METHOD PUBLIC TestTryGetKeyUint
VAR
    jsonDeserializer : JsonDeserializer;
    json : STRING := '{"data":12345}';
    out : UINT;
	feedback : DeserializerFeedback;
    expected : UINT := 12345;
END_VAR
TEST('TestTryGetKeyUint');

jsonDeserializer.TryLoad(json);
jsonDeserializer.TryGetKeyUint('data', out, feedback);

AssertEquals(
    Expected := expected,
    Actual := out,
    Message := 'Did not produce the expected UINT value from JSON'
);

TEST_FINISHED();
END_METHOD

METHOD PUBLIC TestTryGetKeyUlint
VAR
    jsonDeserializer : JsonDeserializer;
    json : STRING := '{"data":9223372036854775807}';
    out : ULINT;
	feedback : DeserializerFeedback;
    expected : ULINT := 9223372036854775807;
END_VAR
TEST('TestTryGetKeyUlint');

jsonDeserializer.TryLoad(json);
jsonDeserializer.TryGetKeyUlint('data', out, feedback);

AssertEquals(
    Expected := expected,
    Actual := out,
    Message := 'Did not produce the expected ULINT value from JSON'
);

TEST_FINISHED();
END_METHOD

METHOD PUBLIC TestTryGetKeyUsint
VAR
    jsonDeserializer : JsonDeserializer;
    json : STRING := '{"data":123}';
    out : USINT;
	feedback : DeserializerFeedback;
    expected : USINT := 123;
END_VAR
TEST('TestTryGetKeyUsint');

jsonDeserializer.TryLoad(json);
jsonDeserializer.TryGetKeyUsint('data', out, feedback);

AssertEquals(
    Expected := expected,
    Actual := out,
    Message := 'Did not produce the expected USINT value from JSON'
);

TEST_FINISHED();
END_METHOD

METHOD PUBLIC TestTryGetKeyWord
VAR
    jsonDeserializer : JsonDeserializer;
    json : STRING := '{"data":12345}';
    out : WORD;
	feedback : DeserializerFeedback;
    expected : WORD := 12345;
END_VAR
TEST('TestTryGetKeyWord');

jsonDeserializer.TryLoad(json);
jsonDeserializer.TryGetKeyWord('data', out, feedback);

AssertEquals(
    Expected := expected,
    Actual := out,
    Message := 'Did not produce the expected WORD value from JSON'
);

TEST_FINISHED();
END_METHOD

METHOD PUBLIC TestTryGetLint
VAR
    jsonDeserializer : JsonDeserializer;
    json : STRING := '9223372036854775807';
    out : LINT;
	feedback : DeserializerFeedback;
    expected : LINT := 9223372036854775807;
END_VAR
TEST('TestTryGetLint');

jsonDeserializer.TryLoad(json);
jsonDeserializer.TryGetLint(out, feedback);

AssertEquals(
    Expected := expected,
    Actual := out,
    Message := 'Did not produce the expected LINT value from JSON'
);

TEST_FINISHED();
END_METHOD

METHOD PUBLIC TestTryGetLreal
VAR
    jsonDeserializer : JsonDeserializer;
    json : STRING := '123456.789';
    out : LREAL;
	feedback : DeserializerFeedback;
    expected : LREAL := 123456.789;
END_VAR
TEST('TestTryGetLreal');

jsonDeserializer.TryLoad(json);
jsonDeserializer.TryGetLreal(out, feedback);

AssertEquals(
    Expected := expected,
    Actual := out,
    Message := 'Did not produce the expected LREAL value from JSON'
);

TEST_FINISHED();
END_METHOD

METHOD PUBLIC TestTryGetLtime
VAR
    jsonDeserializer : JsonDeserializer;
    json : STRING := '"LTIME#100d2h30m40s500ms600us700ns"';
    out : LTIME;
	feedback : DeserializerFeedback;
    expected : LTIME := LTIME#100D2H30M40S500MS600US700NS;
END_VAR
TEST('TestTryGetLtime');

jsonDeserializer.TryLoad(json);
jsonDeserializer.TryGetLtime(out, feedback);

AssertEquals(
    Expected := expected,
    Actual := out,
    Message := 'Did not produce the expected LTIME value from JSON string'
);

TEST_FINISHED();
END_METHOD

METHOD PUBLIC TestTryGetLword
VAR
    jsonDeserializer : JsonDeserializer;
    json : STRING := '9223372036854775807';
    out : LWORD;
	feedback : DeserializerFeedback;
    expected : LWORD := 9223372036854775807;
END_VAR
TEST('TestTryGetLword');

jsonDeserializer.TryLoad(json);
jsonDeserializer.TryGetLword(out, feedback);

AssertEquals(
    Expected := expected,
    Actual := out,
    Message := 'Did not produce the expected LWORD value from JSON'
);

TEST_FINISHED();
END_METHOD

METHOD PUBLIC TestTryGetReal
VAR
    jsonDeserializer : JsonDeserializer;
    json : STRING := '123.4';
    out : REAL;
	feedback : DeserializerFeedback;
    expected : REAL := 123.4;
END_VAR
TEST('TestTryGetReal');

jsonDeserializer.TryLoad(json);
jsonDeserializer.TryGetReal(out, feedback);

AssertEquals(
    Expected := expected,
    Actual := out,
    Message := 'Did not produce the expected REAL value from JSON'
);

TEST_FINISHED();
END_METHOD

METHOD PUBLIC TestTryGetSint
VAR
    jsonDeserializer : JsonDeserializer;
    json : STRING := '123';
    out : SINT;
	feedback : DeserializerFeedback;
    expected : SINT := 123;
END_VAR
TEST('TestTryGetSint');

jsonDeserializer.TryLoad(json);
jsonDeserializer.TryGetSint(out, feedback);

AssertEquals(
    Expected := expected,
    Actual := out,
    Message := 'Did not produce the expected SINT value from JSON'
);

TEST_FINISHED();
END_METHOD

METHOD PUBLIC TestTryGetString
VAR
    jsonDeserializer : JsonDeserializer;
    json : STRING := '"foobar"';
    out : STRING;
	feedback : DeserializerFeedback;
    expected : STRING := 'foobar';
END_VAR
TEST('TestTryGetString');

jsonDeserializer.TryLoad(json);
jsonDeserializer.TryGetString(out, feedback);

AssertEquals(
    Expected := expected,
    Actual := out,
    Message := 'Did not produce the expected STRING value from JSON "foobar"'
);

TEST_FINISHED();
END_METHOD

METHOD PUBLIC TestTryGetTime
VAR
    jsonDeserializer : JsonDeserializer;
    json : STRING := '"T#49d17h2m47s295ms"';
    out : TIME;
	feedback : DeserializerFeedback;
    expected : TIME := T#49D17H2M47S295MS;
END_VAR
TEST('TestTryGetTime');

jsonDeserializer.TryLoad(json);
jsonDeserializer.TryGetTime(out, feedback);

AssertEquals(
    Expected := expected,
    Actual := out,
    Message := 'Did not produce the expected TIME value from JSON'
);

TEST_FINISHED();
END_METHOD

METHOD PUBLIC TestTryGetTod
VAR
    jsonDeserializer : JsonDeserializer;
    json : STRING := '"TOD#23:01:23.456"';
    out : TOD;
	feedback : DeserializerFeedback;
    expected : TOD := TOD#23:01:23.456;
END_VAR
TEST('TestTryGetTod');

jsonDeserializer.TryLoad(json);
jsonDeserializer.TryGetTod(out, feedback);

AssertEquals(
    Expected := expected,
    Actual := out,
    Message := 'Did not produce the expected TOD value from JSON string'
);

TEST_FINISHED();
END_METHOD

METHOD PUBLIC TestTryGetUdint
VAR
    jsonDeserializer : JsonDeserializer;
    json : STRING := '123456';
    out : UDINT;
	feedback : DeserializerFeedback;
    expected : UDINT := 123456;
END_VAR
TEST('TestTryGetUdint');

jsonDeserializer.TryLoad(json);
jsonDeserializer.TryGetUdint(out, feedback);

AssertEquals(
    Expected := expected,
    Actual := out,
    Message := 'Did not produce the expected UDINT value from JSON'
);

TEST_FINISHED();
END_METHOD

METHOD PUBLIC TestTryGetUint
VAR
    jsonDeserializer : JsonDeserializer;
    json : STRING := '12345';
    out : UINT;
	feedback : DeserializerFeedback;
    expected : UINT := 12345;
END_VAR
TEST('TestTryGetUint');

jsonDeserializer.TryLoad(json);
jsonDeserializer.TryGetUint(out, feedback);

AssertEquals(
    Expected := expected,
    Actual := out,
    Message := 'Did not produce the expected UINT value from JSON'
);

TEST_FINISHED();
END_METHOD

METHOD PUBLIC TestTryGetUlint
VAR
    jsonDeserializer : JsonDeserializer;
    json : STRING := '9223372036854775807';
    out : ULINT;
	feedback : DeserializerFeedback;
    expected : ULINT := 9223372036854775807;
END_VAR
TEST('TestTryGetUlint');

jsonDeserializer.TryLoad(json);
jsonDeserializer.TryGetUlint(out, feedback);

AssertEquals(
    Expected := expected,
    Actual := out,
    Message := 'Did not produce the expected ULINT value from JSON'
);

TEST_FINISHED();
END_METHOD

METHOD PUBLIC TestTryGetUsint
VAR
    jsonDeserializer : JsonDeserializer;
    json : STRING := '123';
    out : USINT;
	feedback : DeserializerFeedback;
    expected : USINT := 123;
END_VAR
TEST('TestTryGetUsint');

jsonDeserializer.TryLoad(json);
jsonDeserializer.TryGetUsint(out, feedback);

AssertEquals(
    Expected := expected,
    Actual := out,
    Message := 'Did not produce the expected USINT value from JSON'
);

TEST_FINISHED();
END_METHOD

METHOD PUBLIC TestTryGetWord
VAR
    jsonDeserializer : JsonDeserializer;
    json : STRING := '12345';
    out : WORD;
	feedback : DeserializerFeedback;
    expected : WORD := 12345;
END_VAR
TEST('TestTryGetWord');

jsonDeserializer.TryLoad(json);
jsonDeserializer.TryGetWord(out, feedback);

AssertEquals(
    Expected := expected,
    Actual := out,
    Message := 'Did not produce the expected WORD value from JSON "12345"'
);

TEST_FINISHED();
END_METHOD

END_FUNCTION_BLOCK

// ---- Tests/Mocks/MockDeserializableUserObject.TcPOU
FUNCTION_BLOCK MockDeserializableUserObject IMPLEMENTS I_Deserializable
VAR
	_name : STRING;
	_age : INT;
END_VAR

PROPERTY PUBLIC Age : INT
GET
Age := _age;
END_GET
SET
_age := Age;
END_SET
END_PROPERTY

METHOD PRIVATE CreateMissingKeyError : I_Error
VAR_INPUT
END_VAR
END_METHOD

PROPERTY PUBLIC Name : STRING
GET
Name := _name;
END_GET
SET
_name := Name;
END_SET
END_PROPERTY

METHOD TryDeserializeFrom : BOOL
VAR_INPUT
	Deserializer : I_Deserializer;
	Feedback : I_DeserializerFeedback;
END_VAR
IF NOT Deserializer.TryGetKeyString('Name',_name, Feedback) THEN
	RETURN;
END_IF

IF NOT Deserializer.TryGetKeyInt('Age',_age, Feedback) THEN
	RETURN;
END_IF

TryDeserializeFrom := TRUE;
END_METHOD

END_FUNCTION_BLOCK

// ---- Tests/JsonDeserializerArrayForwardEnumerator_TestSuite.TcPOU
FUNCTION_BLOCK JsonDeserializerArrayForwardEnumerator_TestSuite EXTENDS TcUnit.FB_TestSuite
VAR
END_VAR

TestIsValidAtStart();
TestIsNotValidAfterParentReset();
TestMoveNextReturnsFalseAtTheEnd();
TestMoveNextReturnsTrueSingleItem();
TestMoveNextReturnsFalseWhenEmpty();
TestMoveNextReturnsTrueMultipleItems();
TestEnumerateThroughArrayOfInts();
TestEnumerateThroughArrayOfStrings();
TestEnumerateThroughArrayOfObjects();

METHOD PRIVATE TestEnumerateThroughArrayOfInts
VAR
	jsonDeserializer : JsonDeserializer;
	enumerator : I_DeserializerArrayForwardEnumerator;
    json : STRING := '[1, 2, 3]';
	out1, out2, out3 : INT;
	feedback1, feedback2, feedback3 : DeserializerFeedback;
	expected1 : INT := 1;
	expected2 : INT := 2;
	expected3 : INT := 3;
	result : BOOL;
END_VAR
TEST('TestEnumerateThroughArrayOfInts');

jsonDeserializer.TryLoad(json);
enumerator := jsonDeserializer.GetArrayEnumerator();

enumerator.MoveNext();
enumerator.Current.TryGetInt(out1, feedback1);

enumerator.MoveNext();
enumerator.Current.TryGetInt(out2, feedback2);

enumerator.MoveNext();
enumerator.Current.TryGetInt(out3, feedback3);

enumerator.Dispose();

AssertEquals(
	Expected := expected1,
	Actual := out1,
	Message := 'Did not produce the expected result'
);

AssertEquals(
	Expected := expected2,
	Actual := out2,
	Message := 'Did not produce the expected result'
);

AssertEquals(
	Expected := expected3,
	Actual := out3,
	Message := 'Did not produce the expected result'
);
	
TEST_FINISHED();
END_METHOD

METHOD PRIVATE TestEnumerateThroughArrayOfObjects
VAR
	jsonDeserializer : JsonDeserializer;
	enumerator : I_DeserializerArrayForwardEnumerator;
    json : STRING := '[{"name":"hello"}, {"name":"world"}, {"name":"foobar"}]';
	out1, out2, out3 : STRING;
	feedback1, feedback2, feedback3 : DeserializerFeedback;
	expected1 : STRING := 'hello';
	expected2 : STRING := 'world';
	expected3 : STRING := 'foobar';
	result : BOOL;
END_VAR
TEST('TestEnumerateThroughArrayOfObjects');

jsonDeserializer.TryLoad(json);
enumerator := jsonDeserializer.GetArrayEnumerator();

enumerator.MoveNext();
enumerator.Current.TryGetKeyString('name', out1, feedback1);

enumerator.MoveNext();
enumerator.Current.TryGetKeyString('name', out2, feedback2);

enumerator.MoveNext();
enumerator.Current.TryGetKeyString('name', out3, feedback3);

enumerator.Dispose();

AssertEquals(
	Expected := expected1,
	Actual := out1,
	Message := 'Did not produce the expected result'
);

AssertEquals(
	Expected := expected2,
	Actual := out2,
	Message := 'Did not produce the expected result'
);

AssertEquals(
	Expected := expected3,
	Actual := out3,
	Message := 'Did not produce the expected result'
);
	
TEST_FINISHED();
END_METHOD

METHOD PRIVATE TestEnumerateThroughArrayOfStrings
VAR
	jsonDeserializer : JsonDeserializer;
	enumerator : I_DeserializerArrayForwardEnumerator;
    json : STRING := '["one", "two", "three"]';
	out1, out2, out3 : STRING;
	feedback1, feedback2, feedback3 : DeserializerFeedback;
	expected1 : STRING := 'one';
	expected2 : STRING := 'two';
	expected3 : STRING := 'three';
	result : BOOL;
END_VAR
TEST('TestEnumerateThroughArrayOfStrings');

jsonDeserializer.TryLoad(json);
enumerator := jsonDeserializer.GetArrayEnumerator();

enumerator.MoveNext();
enumerator.Current.TryGetString(out1, feedback1);

enumerator.MoveNext();
enumerator.Current.TryGetString(out2, feedback2);

enumerator.MoveNext();
enumerator.Current.TryGetString(out3, feedback3);

enumerator.Dispose();

AssertEquals(
	Expected := expected1,
	Actual := out1,
	Message := 'Did not produce the expected result'
);

AssertEquals(
	Expected := expected2,
	Actual := out2,
	Message := 'Did not produce the expected result'
);

AssertEquals(
	Expected := expected3,
	Actual := out3,
	Message := 'Did not produce the expected result'
);
	
TEST_FINISHED();
END_METHOD

METHOD PRIVATE TestIsNotValidAfterParentReset
VAR
	jsonDeserializer : JsonDeserializer;
	enumerator : I_DeserializerArrayForwardEnumerator;
	result : BOOL;
END_VAR
TEST('TestIsNotValidAfterParentReset');

enumerator := jsonDeserializer.GetArrayEnumerator();

jsonDeserializer.Reset();
result := enumerator.IsValid;

enumerator.Dispose();

AssertFalse(
	Condition := result,
	Message := 'IsValid incorrectly returned true after parent was reset'
);

TEST_FINISHED();
END_METHOD

METHOD PRIVATE TestIsValidAtStart
VAR
	jsonDeserializer : JsonDeserializer;
	enumerator : I_DeserializerArrayForwardEnumerator;
	result : BOOL;
END_VAR
TEST('TestIsValidAtStart');

enumerator := jsonDeserializer.GetArrayEnumerator();

result := enumerator.IsValid;
enumerator.Dispose();

AssertTrue(
	Condition := result,
	Message := 'IsValid returned false'
);

TEST_FINISHED();
END_METHOD

METHOD PRIVATE TestMoveNextReturnsFalseAtTheEnd
VAR
	jsonDeserializer : JsonDeserializer;
	enumerator : I_DeserializerArrayForwardEnumerator;
    json : STRING := '[100]';
	result : BOOL;
END_VAR
TEST('CheckMoveNextReturnsFalseAtTheEnd');

jsonDeserializer.TryLoad(json);
enumerator := jsonDeserializer.GetArrayEnumerator();

enumerator.MoveNext();
result := enumerator.MoveNext();

enumerator.Dispose();

AssertFalse(result,
    'MoveNext did not correctly signal the end of the enumeration');
	
TEST_FINISHED();
END_METHOD

METHOD PRIVATE TestMoveNextReturnsFalseWhenEmpty
VAR
	jsonDeserializer : JsonDeserializer;
	enumerator : I_DeserializerArrayForwardEnumerator;
    json : STRING := '[]';
	result : BOOL;
END_VAR
TEST('CheckMoveNextReturnsFalseWhenEmpty');

jsonDeserializer.TryLoad(json);
enumerator := jsonDeserializer.GetArrayEnumerator();

result := enumerator.MoveNext();

enumerator.Dispose();

AssertFalse(result,
    'MoveNext did not correctly signal an empty array');
	
TEST_FINISHED();
END_METHOD

METHOD PRIVATE TestMoveNextReturnsTrueMultipleItems
VAR
	jsonDeserializer : JsonDeserializer;
	enumerator : I_DeserializerArrayForwardEnumerator;
    json : STRING := '[true, false, true]';
	result : BOOL;
END_VAR
TEST('CheckMoveNextReturnsTrueMultipleItems');

jsonDeserializer.TryLoad(json);
enumerator := jsonDeserializer.GetArrayEnumerator();

enumerator.MoveNext();
result := enumerator.MoveNext();

enumerator.Dispose();

AssertTrue(
	Condition := result,
	Message := 'MoveNext did not correctly signal there were more items to follow'
);
	
TEST_FINISHED();
END_METHOD

METHOD PRIVATE TestMoveNextReturnsTrueSingleItem
VAR
	jsonDeserializer : JsonDeserializer;
	enumerator : I_DeserializerArrayForwardEnumerator;
    json : STRING := '[100]';
	result : BOOL;
END_VAR
TEST('CheckMoveNextReturnsTrueSingleItem');

jsonDeserializer.TryLoad(json);
enumerator := jsonDeserializer.GetArrayEnumerator();

result := enumerator.MoveNext();

enumerator.Dispose();

AssertTrue(
	Condition := result,
	Message := 'MoveNext did not correctly signal there were more items to follow, i.e. the first item'
);
	
TEST_FINISHED();
END_METHOD

END_FUNCTION_BLOCK

// ---- Tests/JsonDeserializerObjectForwardEnumerator_TestSuite.TcPOU
FUNCTION_BLOCK JsonDeserializerObjectForwardEnumerator_TestSuite EXTENDS TcUnit.FB_TestSuite
VAR
END_VAR

TestIsValidAtStart();
TestIsNotValidAfterParentReset();
TestMoveNextReturnsFalseAtTheEnd();
TestMoveNextReturnsTrueSingleItem();
TestMoveNextReturnsFalseWhenEmpty();
TestMoveNextReturnsTrueMultipleItems();
TestEnumerateThroughKeys();

METHOD PRIVATE TestEnumerateThroughKeys
VAR
	jsonDeserializer : JsonDeserializer;
	enumerator : I_DeserializerObjectForwardEnumerator;
    json : STRING := '{"key1":"value1", "key2":"value2", "key3":"value3"}';
	out1, out2, out3 : STRING;
	expected1 : STRING := 'key1';
	expected2 : STRING := 'key2';
	expected3 : STRING := 'key3';
	result : BOOL;
END_VAR
TEST('TestEnumerateThroughKeys');

jsonDeserializer.TryLoad(json);
enumerator := jsonDeserializer.GetObjectEnumerator();

enumerator.MoveNext();
out1 := enumerator.Key;

enumerator.MoveNext();
out2 := enumerator.Key;

enumerator.MoveNext();
out3 := enumerator.Key;

enumerator.Dispose();

AssertEquals(
	Expected := expected1,
	Actual := out1,
	Message := 'Did not produce the expected result'
);

AssertEquals(
	Expected := expected2,
	Actual := out2,
	Message := 'Did not produce the expected result'
);

AssertEquals(
	Expected := expected3,
	Actual := out3,
	Message := 'Did not produce the expected result'
);
	
TEST_FINISHED();
END_METHOD

METHOD PRIVATE TestIsNotValidAfterParentReset
VAR
	jsonDeserializer : JsonDeserializer;
	enumerator : I_DeserializerObjectForwardEnumerator;
	result : BOOL;
END_VAR
TEST('TestIsNotValidAfterParentReset');

enumerator := jsonDeserializer.GetObjectEnumerator();

jsonDeserializer.Reset();
result := enumerator.IsValid;

enumerator.Dispose();

AssertFalse(
	Condition := result,
	Message := 'IsValid incorrectly returned true after parent was reset'
);

TEST_FINISHED();
END_METHOD

METHOD PRIVATE TestIsValidAtStart
VAR
	jsonDeserializer : JsonDeserializer;
	enumerator : I_DeserializerObjectForwardEnumerator;
	result : BOOL;
END_VAR
TEST('TestIsValidAtStart');

enumerator := jsonDeserializer.GetObjectEnumerator();

result := enumerator.IsValid;
enumerator.Dispose();

AssertTrue(
	Condition := result,
	Message := 'IsValid returned false'
);

TEST_FINISHED();
END_METHOD

METHOD PRIVATE TestMoveNextReturnsFalseAtTheEnd
VAR
	jsonDeserializer : JsonDeserializer;
	enumerator : I_DeserializerObjectForwardEnumerator;
    json : STRING := '{"key1":"value1"}';
	result : BOOL;
END_VAR
TEST('CheckMoveNextReturnsFalseAtTheEnd');

jsonDeserializer.TryLoad(json);
enumerator := jsonDeserializer.GetObjectEnumerator();

enumerator.MoveNext();
result := enumerator.MoveNext();

enumerator.Dispose();

AssertFalse(result,
    'MoveNext did not correctly signal the end of the enumeration');
	
TEST_FINISHED();
END_METHOD

METHOD PRIVATE TestMoveNextReturnsFalseWhenEmpty
VAR
	jsonDeserializer : JsonDeserializer;
	enumerator : I_DeserializerObjectForwardEnumerator;
    json : STRING := '{}';
	result : BOOL;
END_VAR
TEST('CheckMoveNextReturnsFalseWhenEmpty');

jsonDeserializer.TryLoad(json);
enumerator := jsonDeserializer.GetObjectEnumerator();

result := enumerator.MoveNext();

enumerator.Dispose();

AssertFalse(result,
    'MoveNext did not correctly signal an empty array');
	
TEST_FINISHED();
END_METHOD

METHOD PRIVATE TestMoveNextReturnsTrueMultipleItems
VAR
	jsonDeserializer : JsonDeserializer;
	enumerator : I_DeserializerObjectForwardEnumerator;
    json : STRING := '{"key1":"value1", "key2":"value2"}';
	result : BOOL;
END_VAR
TEST('CheckMoveNextReturnsTrueMultipleItems');

jsonDeserializer.TryLoad(json);
enumerator := jsonDeserializer.GetObjectEnumerator();

enumerator.MoveNext();
result := enumerator.MoveNext();

enumerator.Dispose();

AssertTrue(
	Condition := result,
	Message := 'MoveNext did not correctly signal there were more items to follow'
);
	
TEST_FINISHED();
END_METHOD

METHOD PRIVATE TestMoveNextReturnsTrueSingleItem
VAR
	jsonDeserializer : JsonDeserializer;
	enumerator : I_DeserializerObjectForwardEnumerator;
    json : STRING := '{"key1":"value1"}';
	result : BOOL;
END_VAR
TEST('CheckMoveNextReturnsTrueSingleItem');

jsonDeserializer.TryLoad(json);
enumerator := jsonDeserializer.GetObjectEnumerator();

result := enumerator.MoveNext();

enumerator.Dispose();

AssertTrue(
	Condition := result,
	Message := 'MoveNext did not correctly signal there were more items to follow, i.e. the first item'
);
	
TEST_FINISHED();
END_METHOD

END_FUNCTION_BLOCK
